# EPICS substitutions: utcaApp/Db/fmc_adc_common.substitutions
file db/scan_task.template {
    {}
}

file db/fmc_adc_common.template {
    {}
}
